INTERFACE ITcoMessenger

(*~
		<docu>
			<summary>
				Adds message of 'debug' category to the message queue.				 
			</summary>		
		</docu>
~*)
METHOD PUBLIC Debug
VAR_INPUT
	(*~
		<docu>
			<summary>
				Arbitrary message string.			 
			</summary>			
		</docu>
	~*)
	Message : STRING(255);
END_VAR
END_METHOD

(*~
		<docu>
			<summary>
				Adds message of 'error' category to the message queue.				 
			</summary>						
		</docu>
~*)
METHOD PUBLIC Error
VAR_INPUT
	(*~
		<docu>
			<summary>
				Arbitrary message string.			 
			</summary>			
		</docu>
	~*)
	Message : STRING(255);
END_VAR
END_METHOD

(*~
		<docu>
			<summary>
				Adds message of 'information' category to the message queue.				 
			</summary>			
		</docu>
~*)
METHOD PUBLIC Info 
VAR_INPUT
	(*~
		<docu>
			<summary>
				Arbitrary message string.			 
			</summary>			
		</docu>
	~*)
	Message : STRING(255);
END_VAR
END_METHOD

(*~
		<docu>
			<summary>
				Adds message of 'notification' category to the message queue.				 
			</summary>				
		</docu>
~*)
METHOD Notify 
VAR_INPUT
	(*~
		<docu>
			<summary>
				Arbitrary message string.			 
			</summary>			
		</docu>
	~*)
	Message : STRING(255);
END_VAR
END_METHOD

(*~
		<docu>
			<summary>
				Adds message of given category to the message queue.				 
			</summary>	
			<returns>Message index.</returns>		
		</docu>
~*)
METHOD PUBLIC Post 
VAR_INPUT
	(*~
		<docu>
			<summary>
				Arbitrary message string.			 
			</summary>			
		</docu>
	~*)
	Message : STRING(255);
	(*~
		<docu>
			<summary>
				Message category.			 
			</summary>			
		</docu>
	~*)
	Category : eMessageCategory;	
END_VAR
END_METHOD

METHOD PostConditionally
VAR_INPUT
	Condition : BOOL;
	Message : STRING(255);
	Category : eMessageCategory;
END_VAR
END_METHOD

(*~
		<docu>
			<summary>
				Adds message of 'programming error' category to the message queue.				 
			</summary>				
		</docu>
~*)
METHOD PUBLIC Programming
VAR_INPUT
	(*~
		<docu>
			<summary>
				Arbitrary message string.			 
			</summary>			
		</docu>
	~*)
	Message : STRING(255);
END_VAR
END_METHOD

(*~
		<docu>
			<summary>
				Adds message of 'trace' category to the message queue.				 
			</summary>					
		</docu>
~*)
METHOD PUBLIC Trace : INT
VAR_INPUT
	(*~
		<docu>
			<summary>
				Arbitrary message string.			 
			</summary>			
		</docu>
	~*)
	Message : STRING(255);
END_VAR
END_METHOD

(*~
		<docu>
			<summary>
				Adds message of 'warning' category to the message queue.				 
			</summary>					
		</docu>
~*)
METHOD PUBLIC Warning 
VAR_INPUT
	(*~
		<docu>
			<summary>
				Arbitrary message string.			 
			</summary>			
		</docu>
	~*)
	Message : STRING(255);
END_VAR
END_METHOD

END_INTERFACE

(* stored: Version 1.1.0.1, ProductVersion 3.1.4024.6
   Itf ITcoMessenger: Id {feb2a157-bddb-4314-a4f2-ca2ae8c2472e}
   Method Debug: Id {294b92e2-bbf2-4b41-9650-e675ae4a6994}
   Method Error: Id {48619612-5323-4338-8cd6-fa7724f01583}
   Method Info: Id {778bca89-ba90-498e-a510-8a52636bd636}
   Method Notify: Id {6586cd0e-da1a-4d66-b068-bc981ab36951}
   Method Post: Id {319e60ac-aec4-4718-8ea8-38486b1fbfb7}
   Method PostConditionally: Id {769bd04b-63c8-4c2c-848e-0e9f5ddd282b}
   Method Programming: Id {cfbee919-5f05-4549-97b8-0a313d179cec}
   Method Trace: Id {e6c89fb1-5c65-4bf9-b3e5-3133fdf78d64}
   Method Warning: Id {771b212c-af9e-4d7b-b873-a59b90d31d11} *)
